% RSLogix 500 project X-Axis.RSS, saved by version 8.30.00.16 %
PROJECT "UNTITLED"    % processor: Bul.1763 MicroLogix 1100 Series B %

PROGRAM FILES
  LAD 2   7 rungs

DATA FILES
  O0 OUTPUT  5 elements
  I1 INPUT  7 elements
  S2 STATUS  66 elements
  B3 BINARY  32 elements
  T4 TIMER  40 elements
  C5 COUNTER  32 elements
  R6 CONTROL  16 elements
  N7 INTEGER  105 elements
  F8 FLOAT  1 elements

LADDER 2
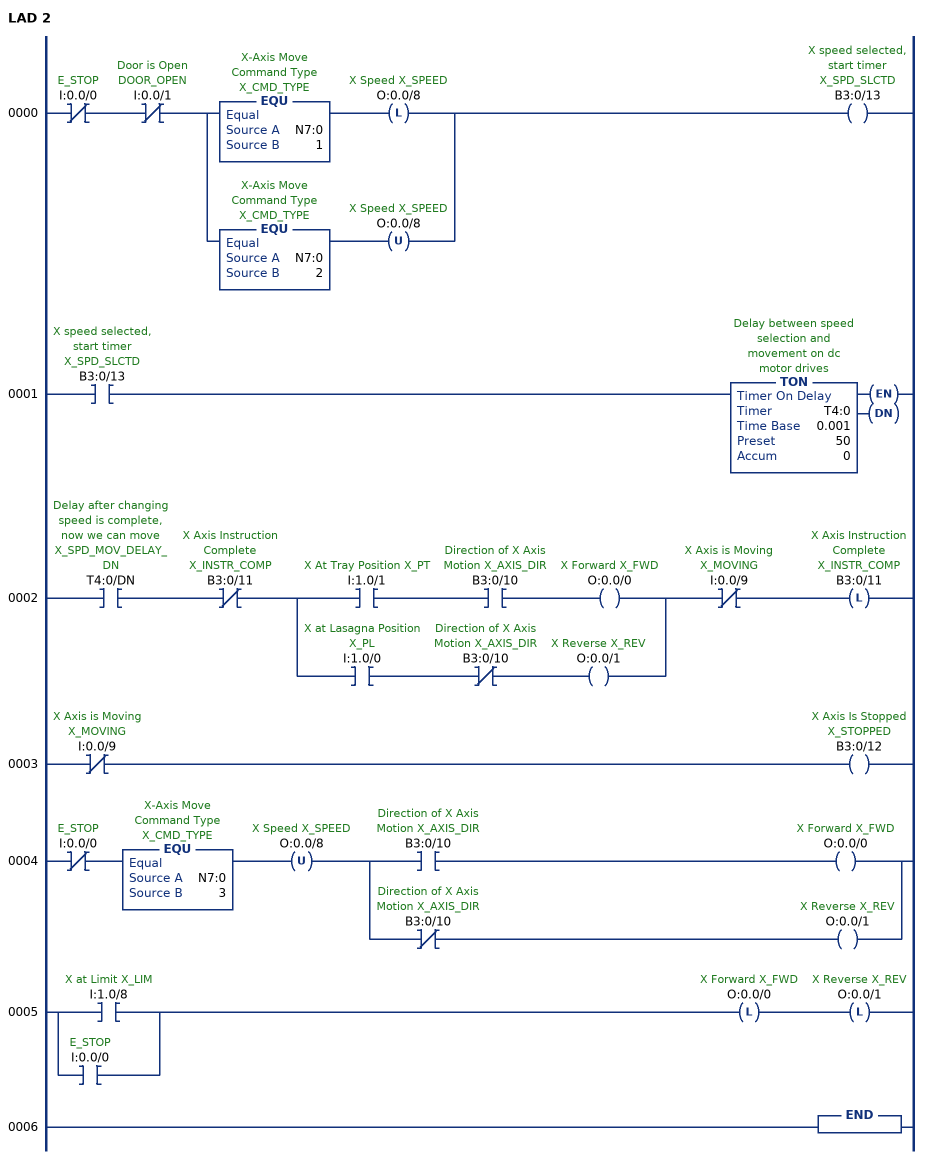
% Rung: 0 %  % edit flag set %
SOR XIO I:0.0/0 XIO I:0.0/1 BST EQU N7:0 1 OTL O:0.0/8 NXB EQU N7:0 2 OTU O:0.0/8 BND OTE B3:0/13 EOR
%   I:0.0/0  E_STOP %
%   I:0.0/1  DOOR_OPEN  "Door is Open" %
%   N7:0  X_CMD_TYPE  "X-Axis Move Command Type" %
%   O:0.0/8  X_SPEED  "X Speed" %
%   B3:0/13  X_SPD_SLCTD  "X speed selected, start timer" %
% Rung: 1 %
SOR XIC B3:0/13 TON T4:0 0.001 50 0 EOR
%   B3:0/13  X_SPD_SLCTD  "X speed selected, start timer" %
%   T4:0  "Delay between speed selection and movement on dc motor drives" %
% Rung: 2 %  % edit flag set %
SOR XIC T4:0/DN XIO B3:0/11 BST XIC I:1.0/1 XIC B3:0/10 OTE O:0.0/0 NXB XIC I:1.0/0 XIO B3:0/10 OTE O:0.0/1 BND XIO I:0.0/9 OTL B3:0/11 EOR
%   T4:0/DN  X_SPD_MOV_DELAY_DN  "Delay after changing speed is complete, now we can move" %
%   B3:0/11  X_INSTR_COMP  "X Axis Instruction Complete" %
%   I:1.0/1  X_PT  "X At Tray Position" %
%   B3:0/10  X_AXIS_DIR  "Direction of X Axis Motion" %
%   O:0.0/0  X_FWD  "X Forward" %
%   I:1.0/0  X_PL  "X at Lasagna Position" %
%   O:0.0/1  X_REV  "X Reverse" %
%   I:0.0/9  X_MOVING  "X Axis is Moving" %
% Rung: 3 %
SOR XIO I:0.0/9 OTE B3:0/12 EOR
%   I:0.0/9  X_MOVING  "X Axis is Moving" %
%   B3:0/12  X_STOPPED  "X Axis Is Stopped" %
% Rung: 4 %  % edit flag set %
SOR XIO I:0.0/0 EQU N7:0 3 OTU O:0.0/8 BST XIC B3:0/10 OTE O:0.0/0 NXB XIO B3:0/10 OTE O:0.0/1 BND EOR
%   I:0.0/0  E_STOP %
%   N7:0  X_CMD_TYPE  "X-Axis Move Command Type" %
%   O:0.0/8  X_SPEED  "X Speed" %
%   B3:0/10  X_AXIS_DIR  "Direction of X Axis Motion" %
%   O:0.0/0  X_FWD  "X Forward" %
%   O:0.0/1  X_REV  "X Reverse" %
% Rung: 5 %  % edit flag set %
SOR BST XIC I:1.0/8 NXB XIC I:0.0/0 BND OTL O:0.0/0 OTL O:0.0/1 EOR
%   I:1.0/8  X_LIM  "X at Limit" %
%   I:0.0/0  E_STOP %
%   O:0.0/0  X_FWD  "X Forward" %
%   O:0.0/1  X_REV  "X Reverse" %
% Rung: 6 %
SOR END EOR

OTHER DOCUMENTED ADDRESSES
  DFILE:0  "OUTPUT"
  DFILE:1  "INPUT"
  DFILE:2  "STATUS"
  DFILE:3  "BINARY"
  DFILE:4  "TIMER"
  DFILE:5  "COUNTER"
  DFILE:6  "CONTROL"
  DFILE:7  "INTEGER"
  DFILE:8  "FLOAT"
  I:1.0/9  "X- Axis Jog Requested ="
  O:0.0/4  X_DIR  "X axis motor direction pin"

DATA TABLE (non-zero values as saved)
DATA T4
% .PRE .ACC %
% T4:0 % 50 0
